FUNCTION_BLOCK fb_eleControllers
VAR_INPUT
END_VAR
VAR_OUTPUT
END_VAR
VAR
END_VAR

gvl_elecylinder.fbi_axisTransport(
	var_ref_ele:= gvl_elecylinder.ref_axis_transport, 
	in_flg_run:= , 
	in_var_moveMode:= , 
	in_flg_pause:= , 
	out_flg_run=> , 
	out_flg_busy=> , 
	out_flg_Done=> , 
	out_flg_error=> );
gvl_elecylinder.fbi_axisSample(
	var_ref_ele:= gvl_elecylinder.ref_axis_sample, 
	in_flg_run:= , 
	in_var_moveMode:= , 
	in_flg_pause:= NOT gvl_io.flg_frontSaftyDoor AND gvl_param.var_currentMode = eP_programMode.auto, 
	out_flg_run=> , 
	out_flg_busy=> , 
	out_flg_Done=> , 
	out_flg_error=> );
gvl_elecylinder.fbi_axisTrayChange(
	var_ref_ele:= gvl_elecylinder.ref_axis_trayChange, 
	in_flg_run:= , 
	in_var_moveMode:= , 
	in_flg_pause:=  NOT gvl_io.flg_frontSaftyDoor AND gvl_param.var_currentMode = eP_programMode.auto, 
	out_flg_run=> , 
	out_flg_busy=> , 
	out_flg_Done=> , 
	out_flg_error=> );
gvl_elecylinder.fbi_axisRotary(
	var_ref_ele:= gvl_elecylinder.ref_axis_rotary, 
	in_flg_run:= , 
	in_var_moveMode:= , 
	in_flg_pause:= , 
	out_flg_run=> , 
	out_flg_busy=> , 
	out_flg_Done=> , 
	out_flg_error=> );
gvl_elecylinder.fbi_gm_axisPickUp(
	var_ref_ele:= gvl_elecylinder.ref_gm_axisPickUp, 
	in_flg_run:= , 
	in_var_moveMode:= , 
	in_flg_pause:= , 
	out_flg_run=> , 
	out_flg_busy=> , 
	out_flg_Done=> , 
	out_flg_error=> );
gvl_elecylinder.fbi_gm_axisTransport(
	var_ref_ele:= gvl_elecylinder.ref_gm_axisTransport, 
	in_flg_run:= , 
	in_var_moveMode:= , 
	in_flg_pause:= , 
	out_flg_run=> , 
	out_flg_busy=> , 
	out_flg_Done=> , 
	out_flg_error=> );
	
IF gvl_elecylinder.ref_axis_trayChange.input.in_flg_sensA THEN
	gvl_param.var_currentTrayPos := 1;
	gvl_visu.var_currentTableMsg := "上段";
ELSIF gvl_elecylinder.ref_axis_trayChange.input.in_flg_sensB THEN
	gvl_param.var_currentTrayPos := 2;
	gvl_visu.var_currentTableMsg := "下段";
ELSE 
	gvl_param.var_currentTrayPos := 0;
	gvl_visu.var_currentTableMsg := "テーブル移動中...";
END_IF

END_FUNCTION_BLOCK

(* stored: Version 1.1.0.1, ProductVersion 3.1.4024.11
   POU fb_eleControllers: Id {ee2a9b3a-1c3d-430d-9a31-a32b100ce462}, SpecialFunc None *)
